// TIA Portal V20 export
DATA_BLOCK "Safetyinterface"   // DB256
// stored: MemoryReserve 100
   VAR
      StackDoor1 : "LER_typefDoorInterface";
      StackDoor2 : "LER_typefDoorInterface";
      StackDoor3 : "LER_typefDoorInterface";
      StackDoor4 : "LER_typefDoorInterface";
      StackDoor5 : "LER_typefDoorInterface";
      StackDoor6 : "LER_typefDoorInterface";
      StackDoor7 : "LER_typefDoorInterface";
      StackDoor8 : "LER_typefDoorInterface";
      StackDoor9 : "LER_typefDoorInterface";
      StackDoor10 : "LER_typefDoorInterface";
      StackDoor11 : "LER_typefDoorInterface";
      StackDoor12 : "LER_typefDoorInterface";
   END_VAR
BEGIN
   StackDoor1.commands.Lock := FALSE;
   StackDoor1.commands.Unlock := FALSE;
   StackDoor1.monitoring.DoorOpen := FALSE;
   StackDoor1.monitoring.DoorClose := TRUE;
   StackDoor1.monitoring.DoorLock := TRUE;
   StackDoor1.monitoring.DoorUnLock := FALSE;
   StackDoor1.configuration.referenceDesignator := WSTRING#'AUTO SPL';
   StackDoor2.commands.Lock := FALSE;
   StackDoor2.commands.Unlock := FALSE;
   StackDoor2.monitoring.DoorOpen := FALSE;
   StackDoor2.monitoring.DoorClose := TRUE;
   StackDoor2.monitoring.DoorLock := TRUE;
   StackDoor2.monitoring.DoorUnLock := FALSE;
   StackDoor2.configuration.referenceDesignator := WSTRING#'U/W MAIN';
   StackDoor3.commands.Lock := FALSE;
   StackDoor3.commands.Unlock := FALSE;
   StackDoor3.monitoring.DoorOpen := FALSE;
   StackDoor3.monitoring.DoorClose := TRUE;
   StackDoor3.monitoring.DoorLock := TRUE;
   StackDoor3.monitoring.DoorUnLock := FALSE;
   StackDoor3.configuration.referenceDesignator := WSTRING#'U/W TOP';
   StackDoor4.commands.Lock := FALSE;
   StackDoor4.commands.Unlock := FALSE;
   StackDoor4.monitoring.DoorOpen := FALSE;
   StackDoor4.monitoring.DoorClose := TRUE;
   StackDoor4.monitoring.DoorLock := TRUE;
   StackDoor4.monitoring.DoorUnLock := FALSE;
   StackDoor4.configuration.referenceDesignator := WSTRING#'U/W BTM';
   StackDoor5.commands.Lock := FALSE;
   StackDoor5.commands.Unlock := FALSE;
   StackDoor5.monitoring.DoorOpen := FALSE;
   StackDoor5.monitoring.DoorClose := TRUE;
   StackDoor5.monitoring.DoorLock := TRUE;
   StackDoor5.monitoring.DoorUnLock := FALSE;
   StackDoor5.configuration.referenceDesignator := WSTRING#'TBL FRNT';
   StackDoor6.commands.Lock := FALSE;
   StackDoor6.commands.Unlock := FALSE;
   StackDoor6.monitoring.DoorOpen := FALSE;
   StackDoor6.monitoring.DoorClose := TRUE;
   StackDoor6.monitoring.DoorLock := TRUE;
   StackDoor6.monitoring.DoorUnLock := FALSE;
   StackDoor6.configuration.referenceDesignator := WSTRING#'WINDER';
   StackDoor7.commands.Lock := FALSE;
   StackDoor7.commands.Unlock := FALSE;
   StackDoor7.monitoring.DoorOpen := FALSE;
   StackDoor7.monitoring.DoorClose := TRUE;
   StackDoor7.monitoring.DoorLock := TRUE;
   StackDoor7.monitoring.DoorUnLock := FALSE;
   StackDoor7.configuration.referenceDesignator := WSTRING#'A-WASTE';
   StackDoor8.commands.Lock := FALSE;
   StackDoor8.commands.Unlock := FALSE;
   StackDoor8.monitoring.DoorOpen := FALSE;
   StackDoor8.monitoring.DoorClose := TRUE;
   StackDoor8.monitoring.DoorLock := TRUE;
   StackDoor8.monitoring.DoorUnLock := FALSE;
   StackDoor8.configuration.referenceDesignator := WSTRING#'TBL REAR';
   StackDoor9.commands.Lock := FALSE;
   StackDoor9.commands.Unlock := FALSE;
   StackDoor9.monitoring.DoorOpen := FALSE;
   StackDoor9.monitoring.DoorClose := TRUE;
   StackDoor9.monitoring.DoorLock := TRUE;
   StackDoor9.monitoring.DoorUnLock := FALSE;
   StackDoor9.configuration.referenceDesignator := WSTRING#'C-WASTE';
   StackDoor10.commands.Lock := FALSE;
   StackDoor10.commands.Unlock := FALSE;
   StackDoor10.monitoring.DoorOpen := FALSE;
   StackDoor10.monitoring.DoorClose := TRUE;
   StackDoor10.monitoring.DoorLock := TRUE;
   StackDoor10.monitoring.DoorUnLock := FALSE;
   StackDoor10.configuration.referenceDesignator := WSTRING#'U/W REAR';
   StackDoor11.commands.Lock := FALSE;
   StackDoor11.commands.Unlock := FALSE;
   StackDoor11.monitoring.DoorOpen := FALSE;
   StackDoor11.monitoring.DoorClose := TRUE;
   StackDoor11.monitoring.DoorLock := TRUE;
   StackDoor11.monitoring.DoorUnLock := FALSE;
   StackDoor11.configuration.referenceDesignator := WSTRING#'';
   StackDoor12.commands.Lock := FALSE;
   StackDoor12.commands.Unlock := FALSE;
   StackDoor12.monitoring.DoorOpen := FALSE;
   StackDoor12.monitoring.DoorClose := TRUE;
   StackDoor12.monitoring.DoorLock := TRUE;
   StackDoor12.monitoring.DoorUnLock := FALSE;
   StackDoor12.configuration.referenceDesignator := WSTRING#'';
END_DATA_BLOCK
